(* PLC project  *)

PROGRAM P
  VAR
    ctr : CTU;
  END_VAR

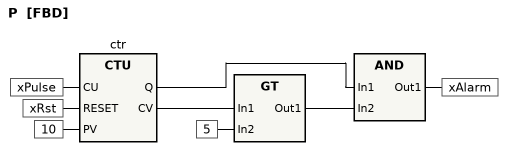
(* FBD diagram, written out as Structured Text *)
ctr(CU := xPulse, RESET := xRst, PV := 10);
xAlarm := ctr.Q AND ctr.CV > 5;
END_PROGRAM
